(* Logix 5000 project; controller PROJECT2 Emulate 5570 rev 30.12; software revision 30.01 *)

TASK MainTask (continuous, watchdog 500 ms) : MainProgram

MODULES
   Local : Emulate 5570 (ICP 0, rev 30.12)
      DC_Input_LIN : vendor 1 type 7 code 2 (ICP 2, rev 2.6, Input RPI 20 ms)
      DC_Output_LOUT : 1756-OB16D (ICP 3, rev 2.3, Output RPI 20 ms)
      Analog_Input : 1756-IF8 (ICP 4, rev 1.5, Input RPI 100 ms)
      HSC : 1756-HSC (ICP 6, rev 1.1, Output RPI 10 ms)
      Analog_Output : 1756-OF4 (ICP 5, rev 1.1, Output RPI 12 ms)
      Devicenet : vendor 1 type 12 code 14 (ICP 7, rev 4.5, Input RPI 20 ms, Output RPI 20 ms)
      EthernetNetwork : vendor 1 type 12 code 200 (ICP 9, Ethernet 192.168.20.11, rev 5.1, Input RPI 500 ms)
         Ethernet3_PointIO : 1734-AENTR (Ethernet 192.168.20.33, rev 5.12, Output RPI 20 ms)
            DCINPUT1 : 1734-IB8 (PointIO 1, rev 3.1)
                 Ethernet3_PointIO:1:I.0   // Walking Beam Clamped
            DCINPUT2 : 1734-IB8 (PointIO 2, rev 3.1)
                 Ethernet3_PointIO:2:I.2   // Station 2 Bottle Filled
            DCINPUT3 : 1734-IB8 (PointIO 3, rev 3.1)
                 Ethernet3_PointIO:3:I.3   // Station 4 Bottle Present
            DCOUTPUT1 : 1734-OB8 (PointIO 4, rev 3.1)
            DCOUTPUT2 : 1734-OB8 (PointIO 5, rev 3.1)
            DCOUTPUT3 : 1734-OB8 (PointIO 6, rev 3.1)
                 Ethernet3_PointIO:6:O.1   // Station 4 Cap Rotate Raised
END_MODULES

TYPE Cylinder :
STRUCT
   DelayTmr : TIMER;
   Complete : BOOL;
   ValveButton : BOOL;
END_STRUCT
END_TYPE

TYPE CylinderExtRet :
STRUCT
   Extend : Cylinder;
   Retract : Cylinder;
END_STRUCT
END_TYPE

TYPE CylinderRaiseLower :
STRUCT
   Raise : Cylinder;
   Lower : Cylinder;
END_STRUCT
END_TYPE

TYPE PartNavigation :
STRUCT
   Directed : BOOL;
   Transferring : BOOL;
   TransferDelay : TIMER;
   Enabled : BOOL;
   Request : BOOL;
   Complete : BOOL;
   EnableTimer : TIMER;
END_STRUCT
END_TYPE

TYPE RandomNumber :
STRUCT
   RandomNum : DINT;
   High : DINT;   // This is a high number 9999999
   Low : DINT;   // This is a low number, ie. 1111111
   Range : DINT;   // This is the upper range of the Random Number
   ONS : BOOL;
   Temp : DINT;
END_STRUCT
END_TYPE

TYPE SIMDoubleCylinder :
STRUCT
   Animation : DINT;
   Extend_ScanCount : DINT;
   Max : DINT;
   Retract_ScanCount : DINT;
   Extend_Timer : TIMER;
   Retract_Timer : TIMER;
   Extend_Output : BOOL;
   Retract_Output : BOOL;
   Extend_Sensor : BOOL;
   Retract_Sensor : BOOL;
   Extend_ValvePB : BOOL;
   Retract_ValvePB : BOOL;
END_STRUCT
END_TYPE

TYPE SIMGeneralSensor :
STRUCT
   ONDelay : TIMER;
   OFFDelay : TIMER;
   ON : BOOL;
   ONCount : COUNTER;
   OFFCount : COUNTER;
   Animation : DINT;
   ONSensingTime : DINT;
   Travelling : BOOL;
   SensingCount : DINT;
   OFFSensingTime : DINT;
   SensingTime : DINT;
END_STRUCT
END_TYPE

TYPE SIMPartTravel :
STRUCT
   Travelling : BOOL;
   Max : DINT;
   Animation : DINT;
   Tmr : TIMER;
   Sensor : BOOL;
   TP_PB : BOOL;
END_STRUCT
END_TYPE

TYPE SIMPartTravelling :
STRUCT
   Enable : BOOL;
   ONS : BOOL;
   EnablePulse : BOOL;
   LiftToPR : SIMPartTravel;
   PrePRtoPR : SIMPartTravel;
   PartRel : SIMPartTravel;
   Reject : SIMPartTravel;
   Divert : SIMPartTravel;
   Conveyor : SIMPartTravel;
   Lift : SIMPartTravel;
   RejectCH : SIMPartTravel;
   DivertCH : SIMPartTravel;
   DivertCONV : SIMPartTravel;
   DivertCONVFlip : SIMPartTravel;
END_STRUCT
END_TYPE

TYPE SIMSingleCylinder :
STRUCT
   Extend_Output : BOOL;
   Extend_ValvePB : BOOL;
END_STRUCT
END_TYPE

TYPE StationStatus :
STRUCT
   BottlePresent : BOOL;
   BottleFilled : BOOL;
   CapInserted : BOOL;
   CapSecured : BOOL;
   TP_FillToggle : BOOL;
   TP_InsertToggle : BOOL;
   TP_SecureToggle : BOOL;
END_STRUCT
END_TYPE

TYPE TouchPanel :
STRUCT
   PLC : TouchPanelPLC;
   Stn : TouchPanelStn;
   Conv : TouchPanelConv;
   Servo : TouchPanelServo;
END_STRUCT
END_TYPE

TYPE TouchPanelConv :
STRUCT
   CurrentPositionIND : REAL;
   TargetSpeed : REAL;
   Fwd : TPBool;
   Rev : TPBool;
   Stop : TPBool;
   Home : TPBool;
   FaultReset : TPBool;
   RemCntl : TouchPanelOnOff;
END_STRUCT
END_TYPE

TYPE TouchPanelExtRet :
STRUCT
   Ext : TPBool;
   Ret : TPBool;
END_STRUCT
END_TYPE

TYPE TouchPanelOnOff :
STRUCT
   On : TPBool;
   Off : TPBool;
END_STRUCT
END_TYPE

TYPE TouchPanelPLC :
STRUCT
   INT1 : INT;
   INT1_TXT : STRING;
   INT2 : INT;
   INT2_TXT : STRING;
   INT3 : INT;
   INT3_TXT : STRING;
   INT4 : INT;
   INT4_TXT : STRING;
   REAL1 : REAL;
   REAL1_TXT : STRING;
   REAL2 : REAL;
   REAL2_TXT : STRING;
   REAL3 : REAL;
   REAL3_TXT : STRING;
   REAL4 : REAL;
   REAL4_TXT : STRING;
   GRAY : TPBool;
   BLUE : TPBool;
   GREEN : TPBool;
   YELLOW : TPBool;
   RED : TPBool;
END_STRUCT
END_TYPE

TYPE TouchPanelRaiseLower :
STRUCT
   Raise : TPBool;
   Lower : TPBool;
END_STRUCT
END_TYPE

TYPE TouchPanelServo :
STRUCT
   Power : TouchPanelOnOff;
   Feedback : TouchPanelOnOff;
   Suction : TouchPanelOnOff;
   Vertical : TouchPanelRaiseLower;
   Home : TPBool;
   CurrentPostionIND : REAL;
   JogSpeed : REAL;
   MoveRight : TPBool;
   MoveLeft : TPBool;
   TargetPosition : REAL;
   TargetSpeed : REAL;
   MoveToTarget : TPBool;
   FaultReset : TPBool;
   Cancel : TPBool;
END_STRUCT
END_TYPE

TYPE TouchPanelStn :
STRUCT
   Auto : TPBool;
   Manual : TPBool;
   CycleStart : TPBool;
   CycleStop : TPBool;
   Lift : TouchPanelRaiseLower;
   PartRelease : TouchPanelOnOff;
   Reject : TouchPanelExtRet;
   Divert : TouchPanelExtRet;
   SendToRejectChute : TPBool;
   SendToDivertChute : TPBool;
   SendToConv : TPBool;
   InsertPart : TPBool;
   FaultReset : TPBool;
END_STRUCT
END_TYPE

TYPE TPBool :
STRUCT
   PB : BOOL;
   PB_TXT : STRING;
   LT : BOOL;
   LT_TXT : STRING;
END_STRUCT
END_TYPE

ADD_ON_INSTRUCTION AOI_SIM_2PosCyl_ExtRet   (* revision 1.0 *)
VAR_INPUT
   TravelTime : DINT; {visible}
END_VAR
VAR_OUTPUT
   Animation : DINT; {visible}
END_VAR
VAR_INPUT
   Extend_Output : BOOL; {required}
   Retract_Output : BOOL; {required}
END_VAR
VAR_OUTPUT
   Extend_Sensor : BOOL; {access Read Only, required}
   Retract_Sensor : BOOL; {access Read Only, required}
END_VAR
VAR_INPUT
   MCR : BOOL; {required}
   SingleSolenoidExtend : BOOL := 1; {required}
   SingleSolenoidRetract : BOOL; {required}
   Retract_ValvePB : BOOL;
   Extend_ValvePB : BOOL;
   DefaultToExt : BOOL; {required}
END_VAR
VAR_OUTPUT
   Extend_Activated : BOOL; {access Read Only}
   Retract_Activated : BOOL; {access Read Only}
END_VAR
VAR
   Extend_ScanCount : DINT;
   Retract_ScanCount : DINT; {access None}
   Extend_Timer : TIMER := (PRE := 500); {access None}
   Retract_Timer : TIMER := (PRE := 500); {access None}
   Retracted : BOOL; {access None}
   Extended : BOOL; {access None}
END_VAR

ROUTINE Logic   (* ladder *)
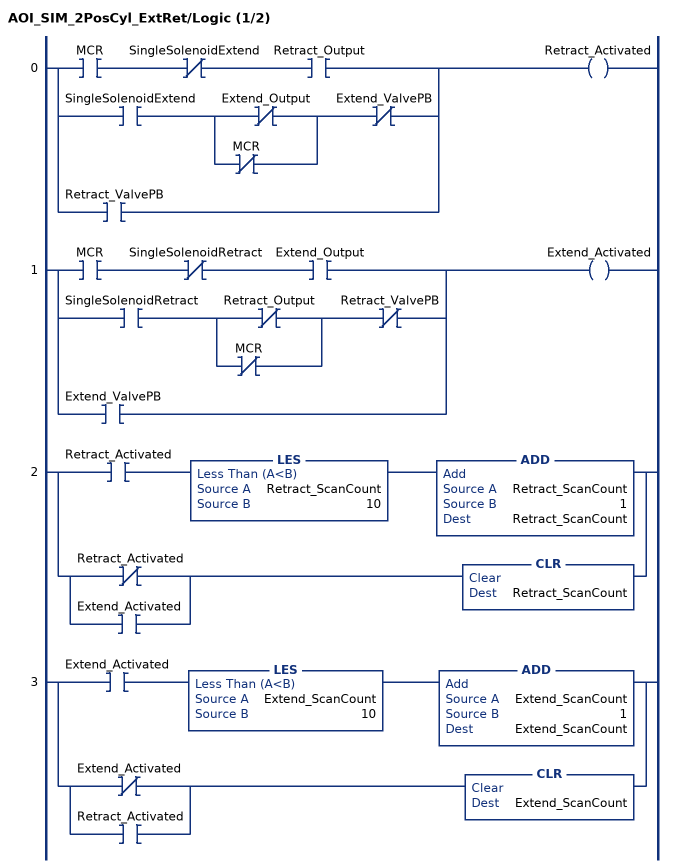
   0: [XIC(MCR) XIO(SingleSolenoidExtend) XIC(Retract_Output) ,XIC(SingleSolenoidExtend) [XIO(Extend_Output) ,XIO(MCR) ] XIO(Extend_ValvePB) ,XIC(Retract_ValvePB) ]OTE(Retract_Activated);
   1: [XIC(MCR) XIO(SingleSolenoidRetract) XIC(Extend_Output) ,XIC(SingleSolenoidRetract) [XIO(Retract_Output) ,XIO(MCR) ] XIO(Retract_ValvePB) ,XIC(Extend_ValvePB) ]OTE(Extend_Activated);
   2: [XIC(Retract_Activated) LES(Retract_ScanCount,10) ADD(Retract_ScanCount,1,Retract_ScanCount) ,[XIO(Retract_Activated) ,XIC(Extend_Activated) ] CLR(Retract_ScanCount) ];
   3: [XIC(Extend_Activated) LES(Extend_ScanCount,10) ADD(Extend_ScanCount,1,Extend_ScanCount) ,[XIO(Extend_Activated) ,XIC(Retract_Activated) ] CLR(Extend_ScanCount) ];
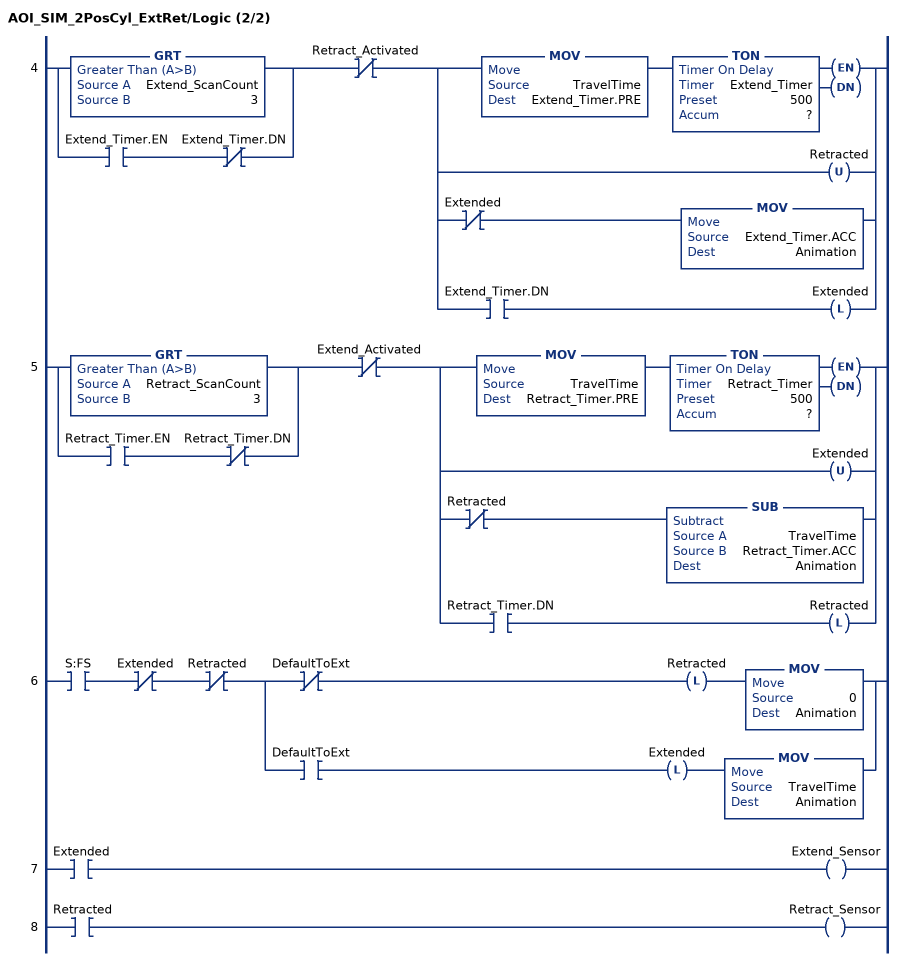
   4: [GRT(Extend_ScanCount,3) ,XIC(Extend_Timer.EN) XIO(Extend_Timer.DN) ]XIO(Retract_Activated)[MOV(TravelTime,Extend_Timer.PRE) TON(Extend_Timer,?,?) ,OTU(Retracted) ,XIO(Extended) MOV(Extend_Timer.ACC,Animation) ,XIC(Extend_Timer.DN) OTL(Extended) ];
   5: [GRT(Retract_ScanCount,3) ,XIC(Retract_Timer.EN) XIO(Retract_Timer.DN) ]XIO(Extend_Activated)[MOV(TravelTime,Retract_Timer.PRE) TON(Retract_Timer,?,?) ,OTU(Extended) ,XIO(Retracted) SUB(TravelTime,Retract_Timer.ACC,Animation) ,XIC(Retract_Timer.DN) OTL(Retracted) ];
   6: XIC(S:FS)XIO(Extended)XIO(Retracted)[XIO(DefaultToExt) OTL(Retracted) MOV(0,Animation) ,XIC(DefaultToExt) OTL(Extended) MOV(TravelTime,Animation) ];
   7: XIC(Extended)OTE(Extend_Sensor);
   8: XIC(Retracted)OTE(Retract_Sensor);
END_ROUTINE
END_ADD_ON_INSTRUCTION

ADD_ON_INSTRUCTION AOI_SIM_2PosCyl_RsLwr   (* revision 1.0 *)
VAR_INPUT
   TravelTime : DINT; {visible}
END_VAR
VAR_OUTPUT
   Animation : DINT; {visible}
END_VAR
VAR_INPUT
   Lower_Output : BOOL; {required}
   Raise_Output : BOOL; {required}
END_VAR
VAR_OUTPUT
   Lower_Sensor : BOOL; {access Read Only, required}
   Raise_Sensor : BOOL; {access Read Only, required}
END_VAR
VAR_INPUT
   MCR : BOOL; {required}
   SingleSolenoidRaise : BOOL; {required}
   SingleSolenoidLower : BOOL; {required}
   Lower_ValvePB : BOOL;
   Raise_ValvePB : BOOL;
   DefaultToLwr : BOOL; {required}
END_VAR
VAR_OUTPUT
   Lower_Activated : BOOL; {access Read Only}
   Raise_Activated : BOOL; {access Read Only}
END_VAR
VAR
   Lower_ScanCount : DINT;
   Raise_ScanCount : DINT; {access None}
   Lower_Timer : TIMER := (PRE := 500); {access None}
   Raise_Timer : TIMER := (PRE := 500); {access None}
   Raised : BOOL; {access None}
   Lowered : BOOL; {access None}
END_VAR

ROUTINE Logic   (* ladder *)
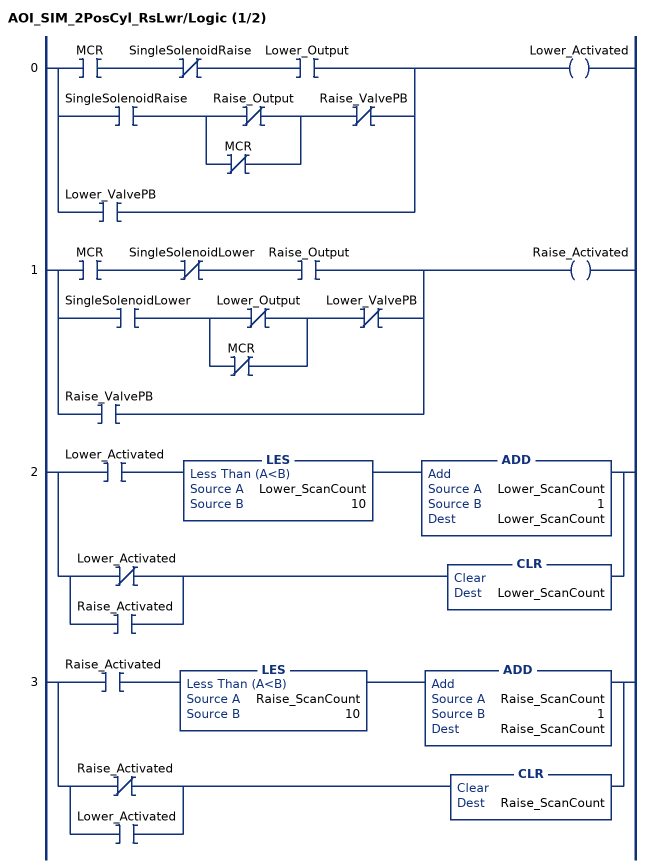
   0: [XIC(MCR) XIO(SingleSolenoidRaise) XIC(Lower_Output) ,XIC(SingleSolenoidRaise) [XIO(Raise_Output) ,XIO(MCR) ] XIO(Raise_ValvePB) ,XIC(Lower_ValvePB) ]OTE(Lower_Activated);
   1: [XIC(MCR) XIO(SingleSolenoidLower) XIC(Raise_Output) ,XIC(SingleSolenoidLower) [XIO(Lower_Output) ,XIO(MCR) ] XIO(Lower_ValvePB) ,XIC(Raise_ValvePB) ]OTE(Raise_Activated);
   2: [XIC(Lower_Activated) LES(Lower_ScanCount,10) ADD(Lower_ScanCount,1,Lower_ScanCount) ,[XIO(Lower_Activated) ,XIC(Raise_Activated) ] CLR(Lower_ScanCount) ];
   3: [XIC(Raise_Activated) LES(Raise_ScanCount,10) ADD(Raise_ScanCount,1,Raise_ScanCount) ,[XIO(Raise_Activated) ,XIC(Lower_Activated) ] CLR(Raise_ScanCount) ];
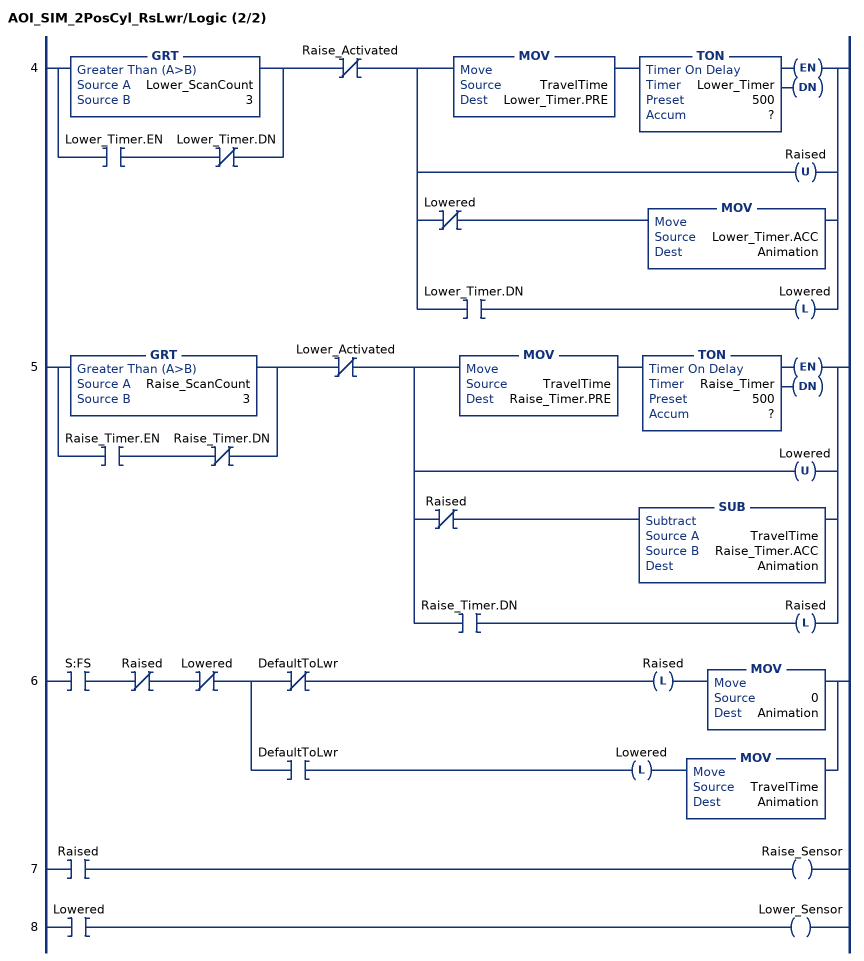
   4: [GRT(Lower_ScanCount,3) ,XIC(Lower_Timer.EN) XIO(Lower_Timer.DN) ]XIO(Raise_Activated)[MOV(TravelTime,Lower_Timer.PRE) TON(Lower_Timer,?,?) ,OTU(Raised) ,XIO(Lowered) MOV(Lower_Timer.ACC,Animation) ,XIC(Lower_Timer.DN) OTL(Lowered) ];
   5: [GRT(Raise_ScanCount,3) ,XIC(Raise_Timer.EN) XIO(Raise_Timer.DN) ]XIO(Lower_Activated)[MOV(TravelTime,Raise_Timer.PRE) TON(Raise_Timer,?,?) ,OTU(Lowered) ,XIO(Raised) SUB(TravelTime,Raise_Timer.ACC,Animation) ,XIC(Raise_Timer.DN) OTL(Raised) ];
   6: XIC(S:FS)XIO(Raised)XIO(Lowered)[XIO(DefaultToLwr) OTL(Raised) MOV(0,Animation) ,XIC(DefaultToLwr) OTL(Lowered) MOV(TravelTime,Animation) ];
   7: XIC(Raised)OTE(Raise_Sensor);
   8: XIC(Lowered)OTE(Lower_Sensor);
END_ROUTINE
END_ADD_ON_INSTRUCTION

ADD_ON_INSTRUCTION AOI_SIM_2PosCyl_RsLwr2pos   (* revision 1.0 *)
VAR_INPUT
   TravelTimeL1 : DINT; {visible}
   TravelTimeL2 : DINT; {visible}
END_VAR
VAR_OUTPUT
   Animation : DINT; {visible}
END_VAR
VAR_INPUT
   Lower_Output : BOOL; {required}
   Raise_Output : BOOL; {required}
END_VAR
VAR_OUTPUT
   Lower1_Sensor : BOOL; {access Read Only, required}
   Lower2_Sensor : BOOL; {access Read Only, required}
END_VAR
VAR_INPUT
   Lower_GoToPos1 : BOOL; {required}
   Lower_GoToPos2 : BOOL; {required}
END_VAR
VAR_OUTPUT
   Raise_Sensor : BOOL; {access Read Only, required}
END_VAR
VAR_INPUT
   MCR : BOOL; {required}
   Lower_ValvePB : BOOL;
   Raise_ValvePB : BOOL;
   DefaultToLwr : BOOL; {required}
END_VAR
VAR
   Raise_ScanCount : DINT; {access None}
   Raise_Timer : TIMER := (PRE := 500); {access None}
   Raised : BOOL; {access None}
   Raise : BOOL; {access None}
   Lowered1 : BOOL; {access None}
   Lower_ScanCount : DINT;
   Lower_Timer : TIMER; {access None}
   Lowered2 : BOOL; {access None}
   Lower : BOOL; {access None}
   RaisePresetONS : BOOL; {access None}
END_VAR

ROUTINE Logic   (* ladder *)
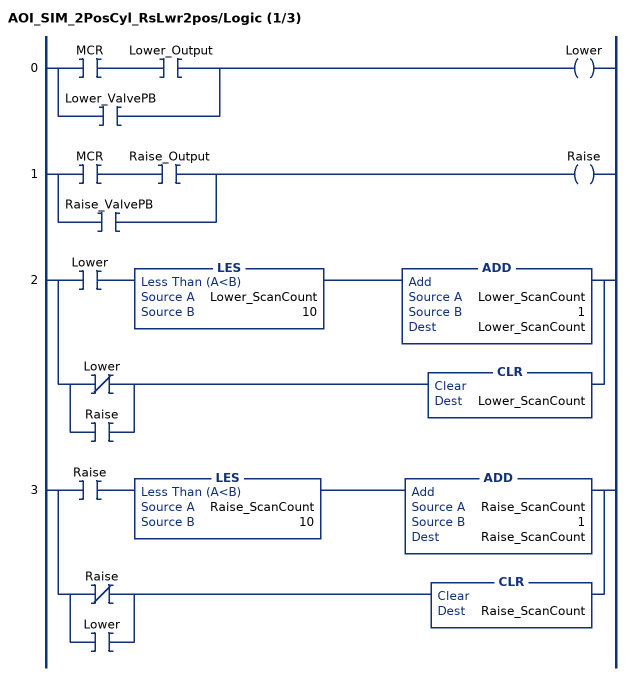
   0: [XIC(MCR) XIC(Lower_Output) ,XIC(Lower_ValvePB) ]OTE(Lower);
   1: [XIC(MCR) XIC(Raise_Output) ,XIC(Raise_ValvePB) ]OTE(Raise);
   2: [XIC(Lower) LES(Lower_ScanCount,10) ADD(Lower_ScanCount,1,Lower_ScanCount) ,[XIO(Lower) ,XIC(Raise) ] CLR(Lower_ScanCount) ];
   3: [XIC(Raise) LES(Raise_ScanCount,10) ADD(Raise_ScanCount,1,Raise_ScanCount) ,[XIO(Raise) ,XIC(Lower) ] CLR(Raise_ScanCount) ];
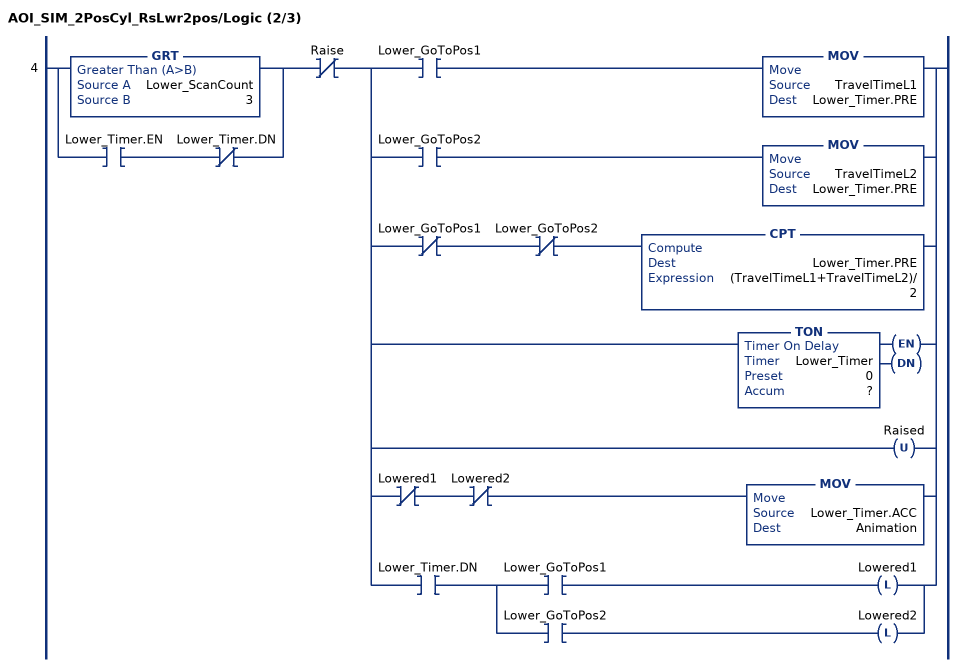
   4: [GRT(Lower_ScanCount,3) ,XIC(Lower_Timer.EN) XIO(Lower_Timer.DN) ]XIO(Raise)[XIC(Lower_GoToPos1) MOV(TravelTimeL1,Lower_Timer.PRE) ,XIC(Lower_GoToPos2) MOV(TravelTimeL2,Lower_Timer.PRE) ,XIO(Lower_GoToPos1) XIO(Lower_GoToPos2) CPT(Lower_Timer.PRE,(TravelTimeL1+TravelTimeL2)/2) ,TON(Lower_Timer,?,?) ,OTU(Raised) ,XIO(Lowered1) XIO(Lowered2) MOV(Lower_Timer.ACC,Animation) ,XIC(Lower_Timer.DN) [XIC(Lower_GoToPos1) OTL(Lowered1) ,XIC(Lower_GoToPos2) OTL(Lowered2) ] ];
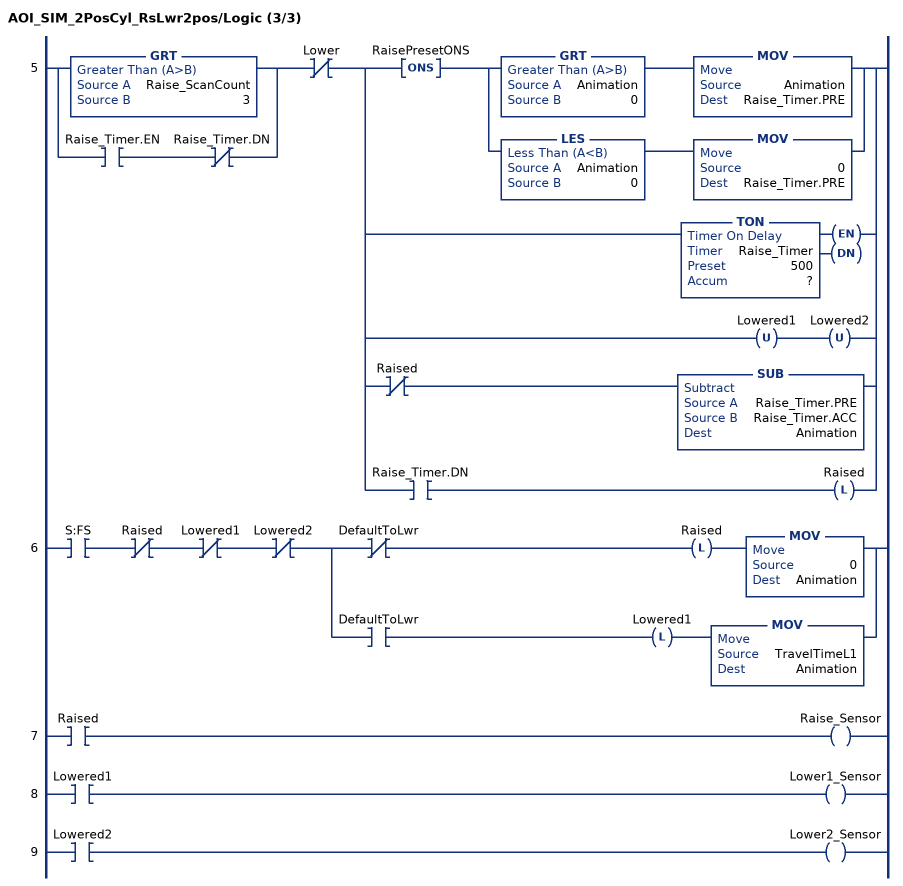
   5: [GRT(Raise_ScanCount,3) ,XIC(Raise_Timer.EN) XIO(Raise_Timer.DN) ]XIO(Lower)[ONS(RaisePresetONS) [GRT(Animation,0) MOV(Animation,Raise_Timer.PRE) ,LES(Animation,0) MOV(0,Raise_Timer.PRE) ] ,TON(Raise_Timer,?,?) ,OTU(Lowered1) OTU(Lowered2) ,XIO(Raised) SUB(Raise_Timer.PRE,Raise_Timer.ACC,Animation) ,XIC(Raise_Timer.DN) OTL(Raised) ];
   6: XIC(S:FS)XIO(Raised)XIO(Lowered1)XIO(Lowered2)[XIO(DefaultToLwr) OTL(Raised) MOV(0,Animation) ,XIC(DefaultToLwr) OTL(Lowered1) MOV(TravelTimeL1,Animation) ];
   7: XIC(Raised)OTE(Raise_Sensor);
   8: XIC(Lowered1)OTE(Lower1_Sensor);
   9: XIC(Lowered2)OTE(Lower2_Sensor);
END_ROUTINE
END_ADD_ON_INSTRUCTION

ADD_ON_INSTRUCTION AOI_SIM_3PosCyl_ExtRet   (* revision 1.0 *)
VAR_INPUT
   TravelTime : DINT; {visible}
END_VAR
VAR_OUTPUT
   Animation : DINT; {visible}
END_VAR
VAR_INPUT
   Extend_Output : BOOL; {required}
   Retract_Output : BOOL; {required}
END_VAR
VAR_OUTPUT
   Extend_Sensor : BOOL; {access Read Only, required}
   Retract_Sensor : BOOL; {access Read Only, required}
END_VAR
VAR_INPUT
   MCR : BOOL; {required}
   Extend_ValvePB : BOOL;
   Retract_ValvePB : BOOL;
   DefaultToExt : BOOL; {required}
END_VAR
VAR_OUTPUT
   Extend_Activated : BOOL; {access Read Only}
   Retract_Activated : BOOL; {access Read Only}
END_VAR
VAR
   Extend_ScanCount : DINT;
   Retract_ScanCount : DINT; {access None}
   Extend_Timer : TIMER := (PRE := 500); {access None}
   Retract_Timer : TIMER := (PRE := 500); {access None}
   Retracted : BOOL; {access None}
   Extended : BOOL; {access None}
   ExtendOneshot : BOOL; {access None}
   RetractOneshot : BOOL; {access None}
END_VAR

ROUTINE Logic   (* ladder *)
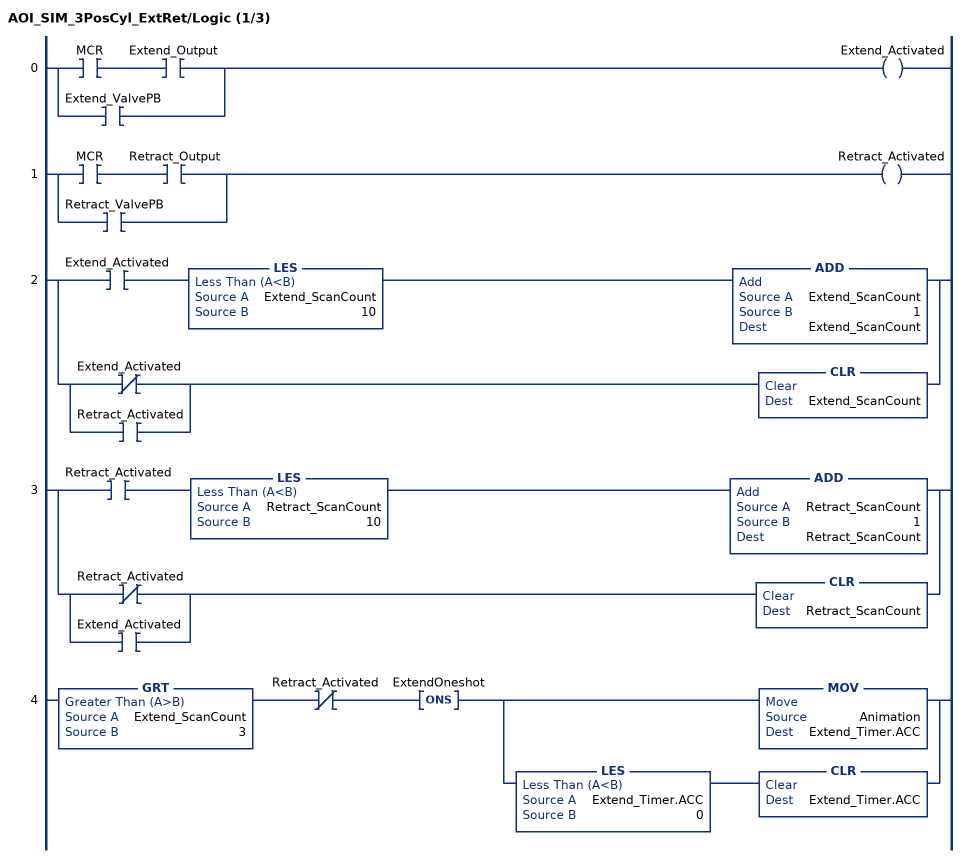
   0: [XIC(MCR) XIC(Extend_Output) ,XIC(Extend_ValvePB) ]OTE(Extend_Activated);
   1: [XIC(MCR) XIC(Retract_Output) ,XIC(Retract_ValvePB) ]OTE(Retract_Activated);
   2: [XIC(Extend_Activated) LES(Extend_ScanCount,10) ADD(Extend_ScanCount,1,Extend_ScanCount) ,[XIO(Extend_Activated) ,XIC(Retract_Activated) ] CLR(Extend_ScanCount) ];
   3: [XIC(Retract_Activated) LES(Retract_ScanCount,10) ADD(Retract_ScanCount,1,Retract_ScanCount) ,[XIO(Retract_Activated) ,XIC(Extend_Activated) ] CLR(Retract_ScanCount) ];
   4: GRT(Extend_ScanCount,3)XIO(Retract_Activated)ONS(ExtendOneshot)[MOV(Animation,Extend_Timer.ACC) ,LES(Extend_Timer.ACC,0) CLR(Extend_Timer.ACC) ];
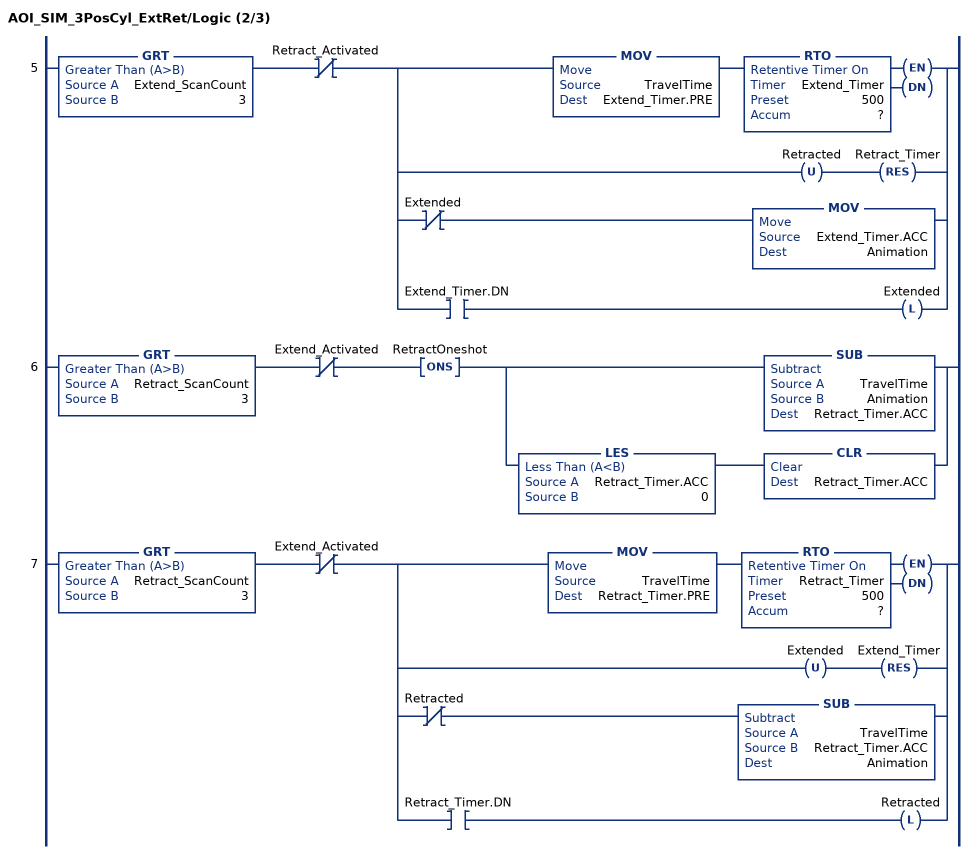
   5: GRT(Extend_ScanCount,3)XIO(Retract_Activated)[MOV(TravelTime,Extend_Timer.PRE) RTO(Extend_Timer,?,?) ,OTU(Retracted) RES(Retract_Timer) ,XIO(Extended) MOV(Extend_Timer.ACC,Animation) ,XIC(Extend_Timer.DN) OTL(Extended) ];
   6: GRT(Retract_ScanCount,3)XIO(Extend_Activated)ONS(RetractOneshot)[SUB(TravelTime,Animation,Retract_Timer.ACC) ,LES(Retract_Timer.ACC,0) CLR(Retract_Timer.ACC) ];
   7: GRT(Retract_ScanCount,3)XIO(Extend_Activated)[MOV(TravelTime,Retract_Timer.PRE) RTO(Retract_Timer,?,?) ,OTU(Extended) RES(Extend_Timer) ,XIO(Retracted) SUB(TravelTime,Retract_Timer.ACC,Animation) ,XIC(Retract_Timer.DN) OTL(Retracted) ];
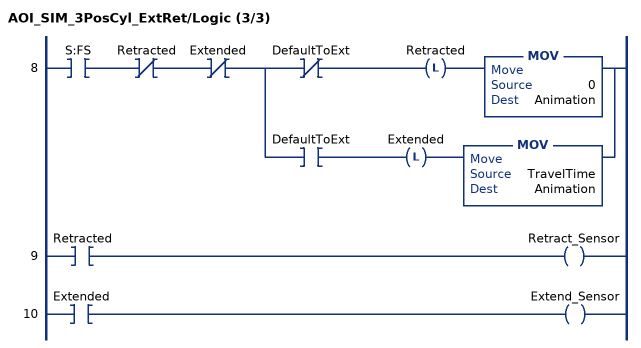
   8: XIC(S:FS)XIO(Retracted)XIO(Extended)[XIO(DefaultToExt) OTL(Retracted) MOV(0,Animation) ,XIC(DefaultToExt) OTL(Extended) MOV(TravelTime,Animation) ];
   9: XIC(Retracted)OTE(Retract_Sensor);
   10: XIC(Extended)OTE(Extend_Sensor);
END_ROUTINE
END_ADD_ON_INSTRUCTION

ADD_ON_INSTRUCTION AOI_SIM_3PosCyl_RsLwr   (* revision 1.0 *)
VAR_INPUT
   TravelTime : DINT; {visible}
END_VAR
VAR_OUTPUT
   Animation : DINT; {visible}
END_VAR
VAR_INPUT
   Lower_Output : BOOL; {required}
   Raise_Output : BOOL; {required}
END_VAR
VAR_OUTPUT
   Lower_Sensor : BOOL; {access Read Only, required}
   Raise_Sensor : BOOL; {access Read Only, required}
END_VAR
VAR_INPUT
   MCR : BOOL; {required}
   Lower_ValvePB : BOOL;
   Raise_ValvePB : BOOL;
   DefaultToLwr : BOOL; {required}
END_VAR
VAR_OUTPUT
   Lower_Activated : BOOL; {access Read Only}
   Raise_Activated : BOOL; {access Read Only}
END_VAR
VAR
   Lower_ScanCount : DINT;
   Raise_ScanCount : DINT; {access None}
   Lower_Timer : TIMER := (PRE := 500); {access None}
   Raise_Timer : TIMER := (PRE := 500); {access None}
   Raised : BOOL; {access None}
   Lowered : BOOL; {access None}
   LowerOneshot : BOOL; {access None}
   RaiseOneshot : BOOL; {access None}
END_VAR

ROUTINE Logic   (* ladder *)
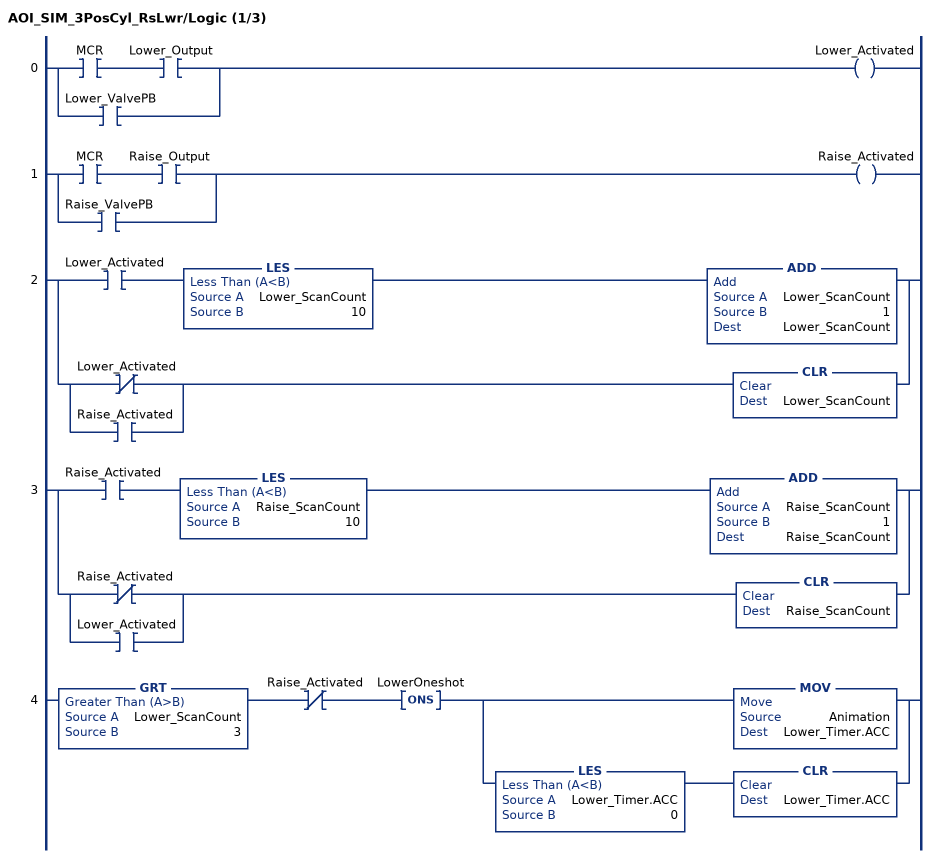
   0: [XIC(MCR) XIC(Lower_Output) ,XIC(Lower_ValvePB) ]OTE(Lower_Activated);
   1: [XIC(MCR) XIC(Raise_Output) ,XIC(Raise_ValvePB) ]OTE(Raise_Activated);
   2: [XIC(Lower_Activated) LES(Lower_ScanCount,10) ADD(Lower_ScanCount,1,Lower_ScanCount) ,[XIO(Lower_Activated) ,XIC(Raise_Activated) ] CLR(Lower_ScanCount) ];
   3: [XIC(Raise_Activated) LES(Raise_ScanCount,10) ADD(Raise_ScanCount,1,Raise_ScanCount) ,[XIO(Raise_Activated) ,XIC(Lower_Activated) ] CLR(Raise_ScanCount) ];
   4: GRT(Lower_ScanCount,3)XIO(Raise_Activated)ONS(LowerOneshot)[MOV(Animation,Lower_Timer.ACC) ,LES(Lower_Timer.ACC,0) CLR(Lower_Timer.ACC) ];
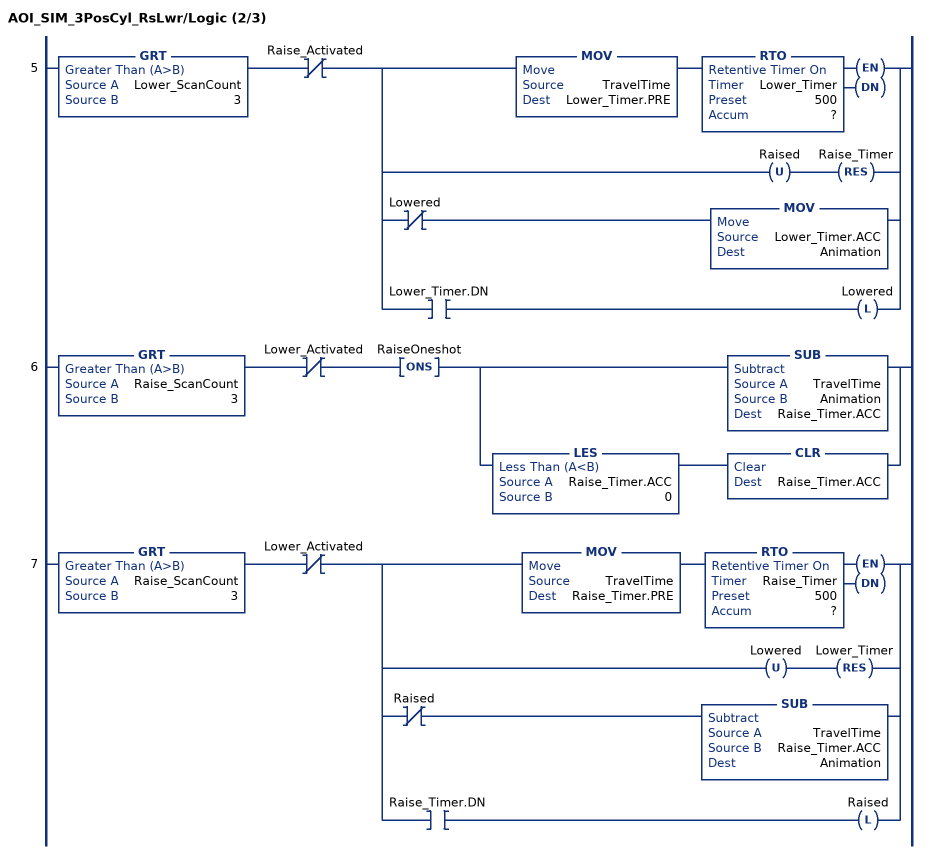
   5: GRT(Lower_ScanCount,3)XIO(Raise_Activated)[MOV(TravelTime,Lower_Timer.PRE) RTO(Lower_Timer,?,?) ,OTU(Raised) RES(Raise_Timer) ,XIO(Lowered) MOV(Lower_Timer.ACC,Animation) ,XIC(Lower_Timer.DN) OTL(Lowered) ];
   6: GRT(Raise_ScanCount,3)XIO(Lower_Activated)ONS(RaiseOneshot)[SUB(TravelTime,Animation,Raise_Timer.ACC) ,LES(Raise_Timer.ACC,0) CLR(Raise_Timer.ACC) ];
   7: GRT(Raise_ScanCount,3)XIO(Lower_Activated)[MOV(TravelTime,Raise_Timer.PRE) RTO(Raise_Timer,?,?) ,OTU(Lowered) RES(Lower_Timer) ,XIO(Raised) SUB(TravelTime,Raise_Timer.ACC,Animation) ,XIC(Raise_Timer.DN) OTL(Raised) ];
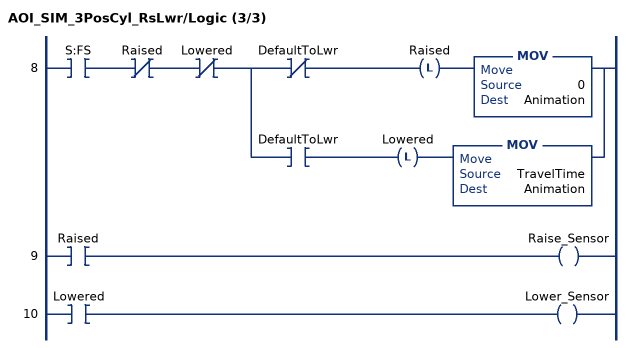
   8: XIC(S:FS)XIO(Raised)XIO(Lowered)[XIO(DefaultToLwr) OTL(Raised) MOV(0,Animation) ,XIC(DefaultToLwr) OTL(Lowered) MOV(TravelTime,Animation) ];
   9: XIC(Raised)OTE(Raise_Sensor);
   10: XIC(Lowered)OTE(Lower_Sensor);
END_ROUTINE
END_ADD_ON_INSTRUCTION

ADD_ON_INSTRUCTION AOI_SIM_Conveyor   (* revision 1.0 *)
VAR_INPUT
   RunDelay : DINT; {visible}
   Output : BOOL; {required}
   MCR : BOOL; {required}
   JogPB : BOOL;
END_VAR
VAR_OUTPUT
   Running : BOOL; {access Read Only, required}
END_VAR
VAR
   Run_ScanCount : DINT;
   Run_Timer : TIMER := (PRE := 500); {access None}
   Run : BOOL; {access None}
END_VAR

ROUTINE Logic   (* ladder *)
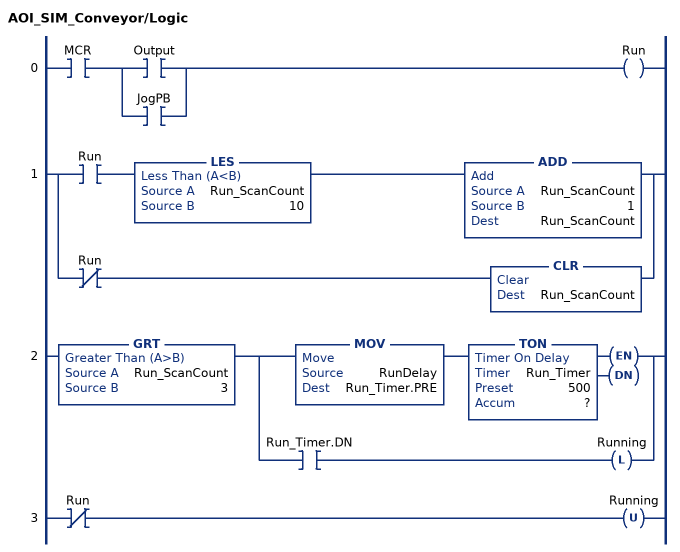
   0: XIC(MCR)[XIC(Output) ,XIC(JogPB) ]OTE(Run);
   1: [XIC(Run) LES(Run_ScanCount,10) ADD(Run_ScanCount,1,Run_ScanCount) ,XIO(Run) CLR(Run_ScanCount) ];
   2: GRT(Run_ScanCount,3)[MOV(RunDelay,Run_Timer.PRE) TON(Run_Timer,?,?) ,XIC(Run_Timer.DN) OTL(Running) ];
   3: XIO(Run)OTU(Running);
END_ROUTINE
END_ADD_ON_INSTRUCTION

ADD_ON_INSTRUCTION AOI_SIM_RandomDelay   (* revision 1.0 *)
VAR_INPUT
   Activate : BOOL; {access None}
   Target : DINT; {access None, visible}
   Tolerance : DINT; {access None, visible}
   PulseOutputTime : DINT; {access None, visible}
END_VAR
VAR_OUTPUT
   DN : BOOL; {access Read Only, required}
END_VAR
VAR_INPUT
   DeActivate : BOOL; {access None}
END_VAR
VAR_OUTPUT
   TimingFirstHalf : BOOL; {access Read Only}
   TimingLastHalf : BOOL; {access Read Only}
   AccumlatedTime : DINT; {access Read Only}
   TT : BOOL; {access Read Only}
END_VAR
VAR
   StartTimerPulse : BOOL; {access None}
   StartTimerONS : BOOL; {access None}
   RandomIntermediate : DINT; {access None}
   RandomNumber : DINT; {access None}
   RandomPresetTime : DINT; {access None}
   RandomTimer : TIMER; {access None}
   PulseOutput : TIMER; {access None}
   Time50Percent : DINT; {access None}
END_VAR

ROUTINE Logic   (* ladder *)
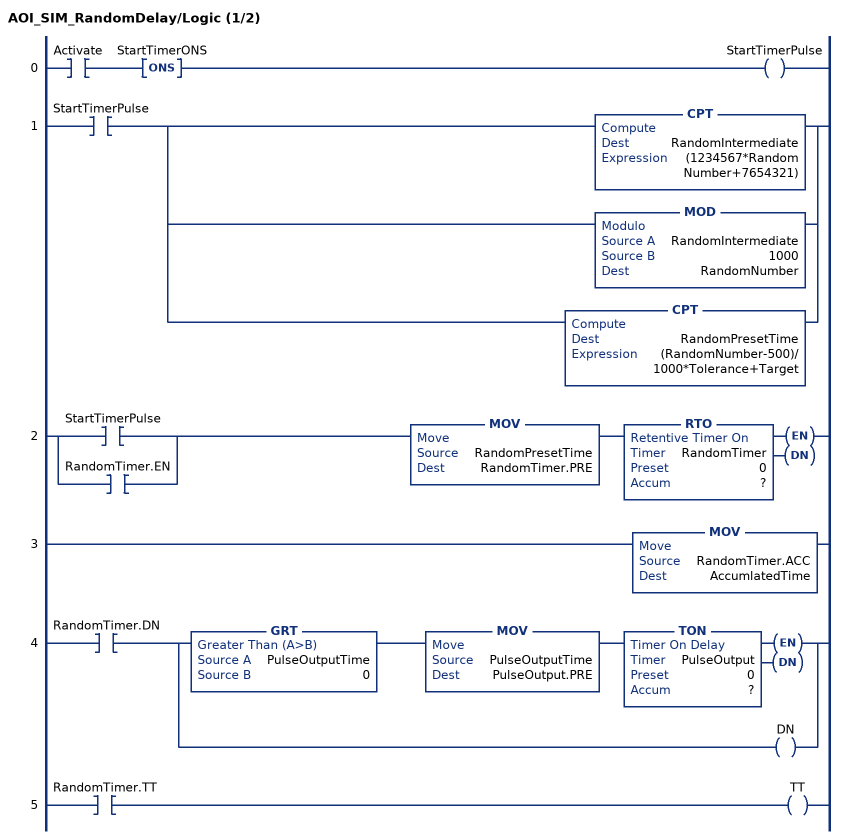
   0: XIC(Activate)ONS(StartTimerONS)OTE(StartTimerPulse);
   1: XIC(StartTimerPulse)[CPT(RandomIntermediate,(1234567*RandomNumber+7654321)) ,MOD(RandomIntermediate,1000,RandomNumber) ,CPT(RandomPresetTime,(RandomNumber-500)/1000*Tolerance+Target) ];
   2: [XIC(StartTimerPulse) ,XIC(RandomTimer.EN) ]MOV(RandomPresetTime,RandomTimer.PRE)RTO(RandomTimer,?,?);
   3: MOV(RandomTimer.ACC,AccumlatedTime);
   4: XIC(RandomTimer.DN)[GRT(PulseOutputTime,0) MOV(PulseOutputTime,PulseOutput.PRE) TON(PulseOutput,?,?) ,OTE(DN) ];
   5: XIC(RandomTimer.TT)OTE(TT);
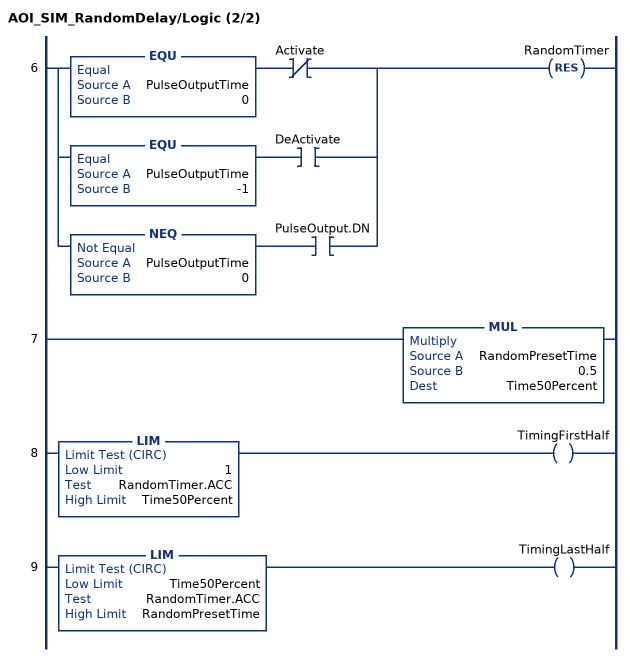
   6: [EQU(PulseOutputTime,0) XIO(Activate) ,EQU(PulseOutputTime,-1) XIC(DeActivate) ,NEQ(PulseOutputTime,0) XIC(PulseOutput.DN) ]RES(RandomTimer);
   7: MUL(RandomPresetTime,0.5,Time50Percent);
   8: LIM(1,RandomTimer.ACC,Time50Percent)OTE(TimingFirstHalf);
   9: LIM(Time50Percent,RandomTimer.ACC,RandomPresetTime)OTE(TimingLastHalf);
END_ROUTINE
END_ADD_ON_INSTRUCTION

ADD_ON_INSTRUCTION AOI_SIM_SimpleValve   (* revision 1.0 *)
VAR_INPUT
   TravelTime : DINT; {visible}
END_VAR
VAR_OUTPUT
   Animation : DINT; {visible}
END_VAR
VAR_INPUT
   Output : BOOL; {required}
   MCR : BOOL; {required}
   ValvePB : BOOL;
END_VAR
VAR_OUTPUT
   Activated : BOOL; {access Read Only}
END_VAR
VAR
   Extend_ScanCount : DINT;
   Retract_ScanCount : DINT; {access None}
   Extend_Timer : TIMER := (PRE := 500); {access None}
   Retract_Timer : TIMER := (PRE := 500); {access None}
   Retracted : BOOL; {access None}
   Extended : BOOL; {access None}
   Retract : BOOL; {access None}
   Extend : BOOL; {access None}
END_VAR

ROUTINE Logic   (* ladder *)
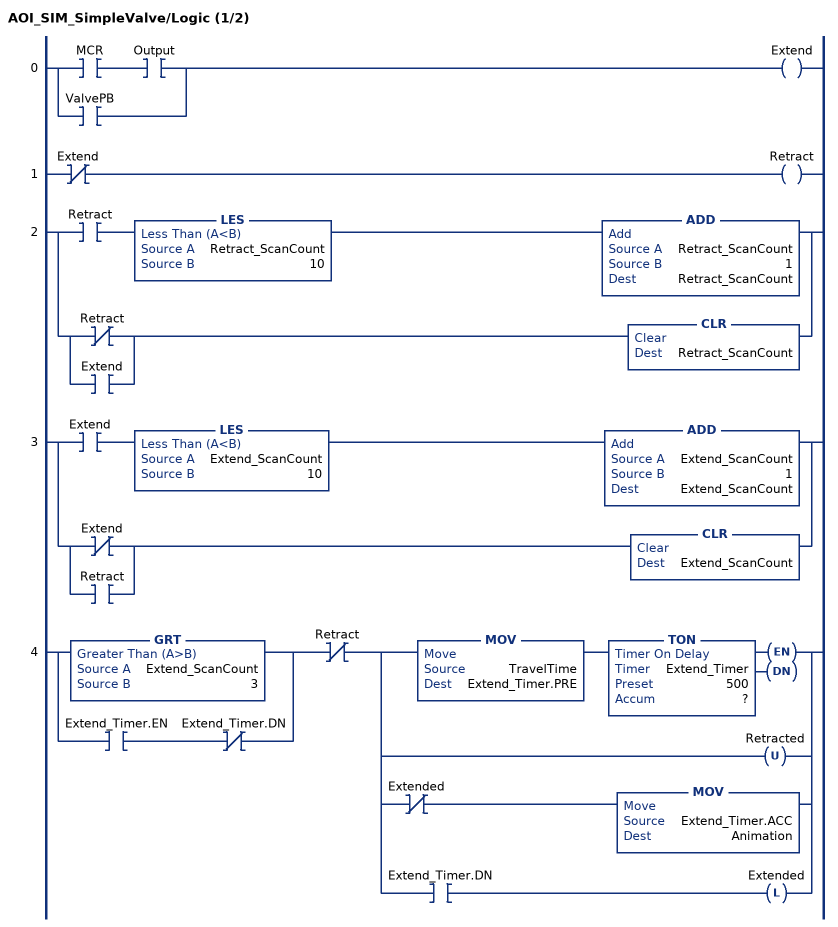
   0: [XIC(MCR) XIC(Output) ,XIC(ValvePB) ]OTE(Extend);
   1: XIO(Extend)OTE(Retract);
   2: [XIC(Retract) LES(Retract_ScanCount,10) ADD(Retract_ScanCount,1,Retract_ScanCount) ,[XIO(Retract) ,XIC(Extend) ] CLR(Retract_ScanCount) ];
   3: [XIC(Extend) LES(Extend_ScanCount,10) ADD(Extend_ScanCount,1,Extend_ScanCount) ,[XIO(Extend) ,XIC(Retract) ] CLR(Extend_ScanCount) ];
   4: [GRT(Extend_ScanCount,3) ,XIC(Extend_Timer.EN) XIO(Extend_Timer.DN) ]XIO(Retract)[MOV(TravelTime,Extend_Timer.PRE) TON(Extend_Timer,?,?) ,OTU(Retracted) ,XIO(Extended) MOV(Extend_Timer.ACC,Animation) ,XIC(Extend_Timer.DN) OTL(Extended) ];
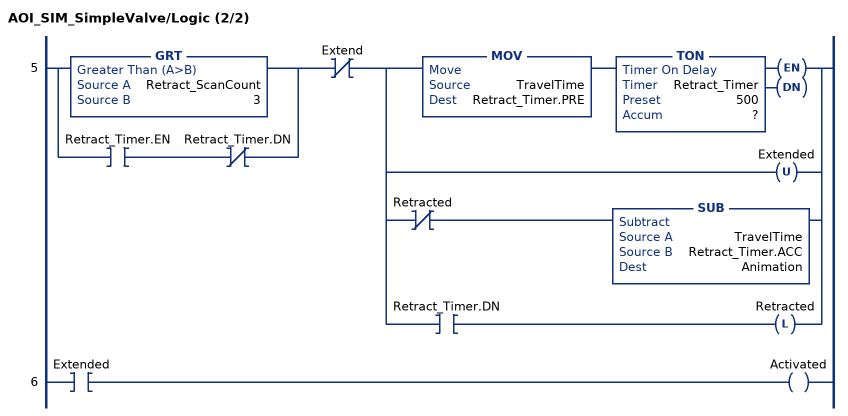
   5: [GRT(Retract_ScanCount,3) ,XIC(Retract_Timer.EN) XIO(Retract_Timer.DN) ]XIO(Extend)[MOV(TravelTime,Retract_Timer.PRE) TON(Retract_Timer,?,?) ,OTU(Extended) ,XIO(Retracted) SUB(TravelTime,Retract_Timer.ACC,Animation) ,XIC(Retract_Timer.DN) OTL(Retracted) ];
   6: XIC(Extended)OTE(Activated);
END_ROUTINE
END_ADD_ON_INSTRUCTION
